FUNCTION_BLOCK ChanSendBool (* Composite Function Block Type *)
  (* Standard: 61499-2 *)
  (* Version 0.0, 7/15/2023, vv263, nxtControl GmBH, template *)
  PACKAGE Main;
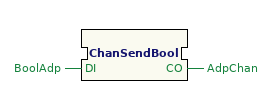
  SOCKETS
    DI : BoolAdp;
  END_SOCKETS
  PLUGS
    CO : AdpChan;
  END_PLUGS
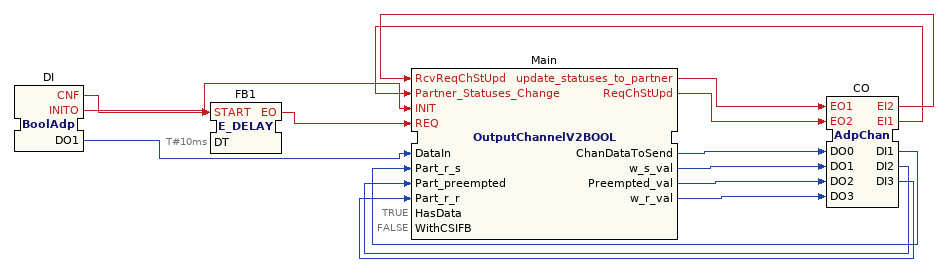
  FBS
    Main : OutputChannelV2BOOL(HasData := TRUE, WithCSIFB := FALSE);
    FB1 : E_DELAY(DT := T#10ms);
  END_FBS
  EVENT_CONNECTIONS
    DI.CNF TO FB1.START;
    Main.update_statuses_to_partner TO CO.EO1;
    Main.ReqChStUpd TO CO.EO2;
    CO.EI2 TO Main.RcvReqChStUpd;
    CO.EI1 TO Main.Partner_Statuses_Change;
    DI.INITO TO Main.INIT;
    FB1.EO TO Main.REQ;
  END_CONNECTIONS
  DATA_CONNECTIONS
    DI.DO1 TO Main.DataIn;
    Main.ChanDataToSend TO CO.DO0;
    Main.w_s_val TO CO.DO1;
    Main.Preempted_val TO CO.DO2;
    Main.w_r_val TO CO.DO3;
    CO.DI1 TO Main.Part_r_s;
    CO.DI2 TO Main.Part_preempted;
    CO.DI3 TO Main.Part_r_r;
  END_CONNECTIONS
END_FUNCTION_BLOCK
